PROGRAM HMI_Invinsible_Ctrl
VAR
	x: BOOL;
	y: BOOL;
END_VAR

//1
IF NOT Global_HMI.bManualOutToUserConfirmPageOn THEN 
	Global_HMI.bManualOutToUserConfirmPageOff:=TRUE;
ELSE
	Global_HMI.bManualOutToUserConfirmPageOff:=FALSE;
END_IF

//2
IF NOT Global_Variables_HMI_Function.bStationOnPage THEN
	Global_Variables_HMI_Function.bStationOffPage :=TRUE;
ELSE
	Global_Variables_HMI_Function.bStationOffPage :=FALSE;
END_IF

//3
IF NOT Global_Variables_HMI_Function.RecipeEditOn THEN
	Global_Variables_HMI_Function.RecipeEditOff :=TRUE;
ELSE
	Global_Variables_HMI_Function.RecipeEditOff :=FALSE;
END_IF

//4
IF NOT NOT Global_HMI.bManualOutToUserConfirmPageOn THEN
	Global_HMI.bManualOutToUserConfirmPageOff :=TRUE;
ELSE
	Global_HMI.bManualOutToUserConfirmPageOff :=FALSE;
END_IF

//5
IF NOT x THEN
	y :=TRUE;
ELSE
	y :=FALSE;
END_IF

//6
IF NOT x THEN
	y :=TRUE;
ELSE
	y :=FALSE;
END_IF

//7
IF NOT x THEN
	y :=TRUE;
ELSE
	y :=FALSE;
END_IF

//8
IF NOT x THEN
	y :=TRUE;
ELSE
	y :=FALSE;
END_IF

//9
IF NOT x THEN
	y :=TRUE;
ELSE
	y :=FALSE;
END_IF

//10
IF NOT x THEN
	y :=TRUE;
ELSE
	y :=FALSE;
END_IF

//11
IF NOT x THEN
	y :=TRUE;
ELSE
	y :=FALSE;
END_IF

//12
IF NOT x THEN
	y :=TRUE;
ELSE
	y :=FALSE;
END_IF

//13
IF NOT x THEN
	y :=TRUE;
ELSE
	y :=FALSE;
END_IF

//14
IF NOT x THEN
	y :=TRUE;
ELSE
	y :=FALSE;
END_IF

//15
IF NOT x THEN
	y :=TRUE;
ELSE
	y :=FALSE;
END_IF

END_PROGRAM

(* stored: Version 1.1.0.1, ProductVersion 3.1.4024.12
   POU HMI_Invinsible_Ctrl: Id {12912e6e-328e-45a2-91c7-84f71ec71d28}, SpecialFunc None *)
